TYPE RegulationControlParameters :
STRUCT
	EN: BOOL := TRUE; // $(W1,S,R0)
	ENO: BOOL;
	StartupHeatRecoveryTime: TIME;
	PostFireVentilationTime: TIME;
	PostVentilationTime: TIME := T#2M;
END_STRUCT
END_TYPE

(* stored: Version 1.1.0.1, ProductVersion 3.1.4024.6
   DUT RegulationControlParameters: Id {ecd9fe89-c947-43c7-96db-b66884bcfdaa} *)
